KUKA KRL data list: drai_gaewint.dat

&ACCESS RVP
&PARAM EDITMASK = *
&PARAM TEMPLATE = C:\KRC\Roboter\Template\ExpertVorgabe
DEFDAT drai_gaewint PUBLIC

ENDDAT
